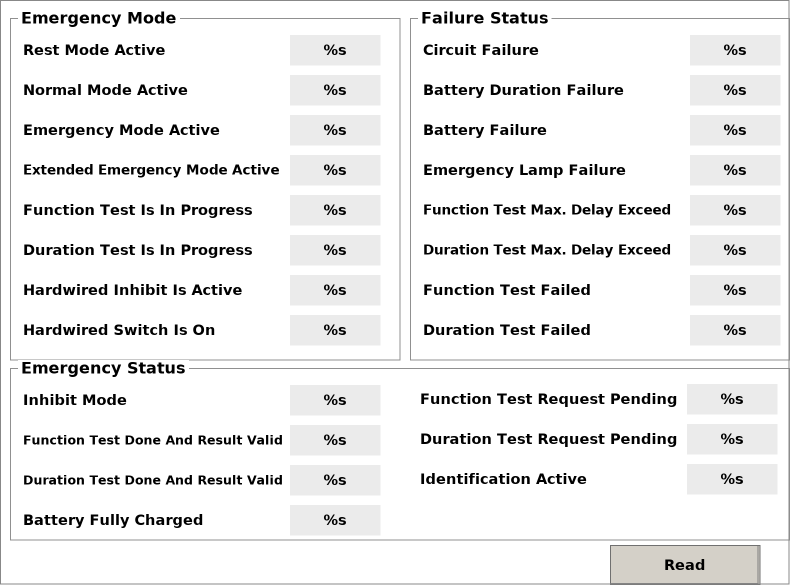
VISUALIZATION Visu_Part202Status  // 790x585
    Button (610,545 150x40), "Read"
        OnMouseClick: execute { DALI_Commissioning.fbPart202Emergency.bReadState:=TRUE; }
    GroupBox (10,10 390x350), "Emergency Mode"
        Textfield (10,145 260x30), "Extended Emergency Mode Active"
        Textfield (280,185 90x30), "%s", text variable: DALI_Commissioning.fbPart202Emergency.sFunctionTest
        Textfield (280,145 90x30), "%s", text variable: DALI_Commissioning.fbPart202Emergency.sExtendedEmergency
        Textfield (280,105 90x30), "%s", text variable: DALI_Commissioning.fbPart202Emergency.sEmergencyMode
        Textfield (280,65 90x30), "%s", text variable: DALI_Commissioning.fbPart202Emergency.sNormalMode
        Textfield (280,25 90x30), "%s", text variable: DALI_Commissioning.fbPart202Emergency.sRestMode
        Textfield (10,25 260x30), "Rest Mode Active"
        Textfield (10,65 260x30), "Normal Mode Active"
        Textfield (10,105 260x30), "Emergency Mode Active"
        Textfield (10,185 260x30), "Function Test Is In Progress"
        Textfield (10,225 260x30), "Duration Test Is In Progress"
        Textfield (10,265 260x30), "Hardwired Inhibit Is Active"
        Textfield (10,305 260x30), "Hardwired Switch Is On"
        Textfield (280,265 90x30), "%s", text variable: DALI_Commissioning.fbPart202Emergency.sHardwiredInhibit
        Textfield (280,305 90x30), "%s", text variable: DALI_Commissioning.fbPart202Emergency.sHardwiredSwitch
        Textfield (280,225 90x30), "%s", text variable: DALI_Commissioning.fbPart202Emergency.sDurationTest
    GroupBox (410,10 380x350), "Failure Status"
        Textfield (10,145 260x30), "Emergency Lamp Failure"
        Textfield (280,185 90x30), "%s", text variable: DALI_Commissioning.fbPart202Emergency.sFunctionTestExceed
        Textfield (280,145 90x30), "%s", text variable: DALI_Commissioning.fbPart202Emergency.sEmergencyLampFailure
        Textfield (280,105 90x30), "%s", text variable: DALI_Commissioning.fbPart202Emergency.sBatteryFailure
        Textfield (280,65 90x30), "%s", text variable: DALI_Commissioning.fbPart202Emergency.sBatteryDurationFailure
        Textfield (280,25 90x30), "%s", text variable: DALI_Commissioning.fbPart202Emergency.sCircuitFailure
        Textfield (10,25 260x30), "Circuit Failure"
        Textfield (10,65 260x30), "Battery Duration Failure"
        Textfield (10,105 260x30), "Battery Failure"
        Textfield (10,185 260x30), "Function Test Max. Delay Exceed"
        Textfield (10,225 260x30), "Duration Test Max. Delay Exceed"
        Textfield (10,265 260x30), "Function Test Failed"
        Textfield (10,305 260x30), "Duration Test Failed"
        Textfield (280,265 90x30), "%s", text variable: DALI_Commissioning.fbPart202Emergency.sFunctionTestFailed
        Textfield (280,305 90x30), "%s", text variable: DALI_Commissioning.fbPart202Emergency.sDurationTestFailed
        Textfield (280,225 90x30), "%s", text variable: DALI_Commissioning.fbPart202Emergency.sDurationTestExceed
    GroupBox (10,360 780x180), "Emergency Status"
        Textfield (10,145 260x30), "Battery Fully Charged"
        Textfield (677,24 90x30), "%s", text variable: DALI_Commissioning.fbPart202Emergency.sFunctionTestRequestPending
        Textfield (10,25 260x30), "Inhibit Mode"
        Textfield (10,65 260x30), "Function Test Done And Result Valid"
        Textfield (407,24 260x30), "Function Test Request Pending"
        Textfield (407,64 260x30), "Duration Test Request Pending"
        Textfield (407,104 260x30), "Identification Active"
        Textfield (677,104 90x30), "%s", text variable: DALI_Commissioning.fbPart202Emergency.sIdentificationActive
        Textfield (677,64 90x30), "%s", text variable: DALI_Commissioning.fbPart202Emergency.sDurationTestRequestPending
        Textfield (280,25 90x30), "%s", text variable: DALI_Commissioning.fbPart202Emergency.sInhibitMode
        Textfield (280,65 90x30), "%s", text variable: DALI_Commissioning.fbPart202Emergency.sFunctionTestDoneValid
        Textfield (280,145 90x30), "%s", text variable: DALI_Commissioning.fbPart202Emergency.sBatteryFullCharged
        Textfield (10,105 260x30), "Duration Test Done And Result Valid"
        Textfield (280,105 90x30), "%s", text variable: DALI_Commissioning.fbPart202Emergency.sDurationTestDoneValid
END_VISUALIZATION

(* stored: Version 1.1.0.1
   Visu Visu_Part202Status: Id {a5e9497f-cce5-4e16-98a8-772d4949a673} *)
